// TIA Portal V17 export
// export: Created 2023-02-25T13:22:14.257017Z, ExportSetting WithDefaults, DisplayName Totally Integrated Automation Portal, DisplayVersion V17, DisplayName TIA Portal Openness, DisplayVersion V17, DisplayName TIA Portal Version Control Interface, DisplayVersion V17, DisplayName TIA Portal Test Suite Advanced, DisplayVersion V17, DisplayName STEP 7 Professional, DisplayVersion V17, DisplayName SIMATIC Energy Suite, DisplayVersion V17, DisplayName STEP 7 Safety, DisplayVersion V17, DisplayName WinCC Professional, DisplayVersion V17
TYPE "stt_Motor"
// stored: IsFailsafeCompliant false
   STRUCT
      Run : Bool;
      LeftTurn : Bool;
      RightTurn : Bool;
      Speed : Real;
   END_STRUCT;
END_TYPE
